FUNCTION_BLOCK xPPU_RFC
VAR_INPUT
	i_error: POINTER TO ErrorManager;
	i_process: POINTER TO ProcessManager;
	i_state: POINTER TO StateTracker;
END_VAR
VAR
	m_emptyParams: ParameterSet;
	m_subRes: EOperationResult;
	m_alarm_flags: ARRAY [1..10] OF BOOL := [FALSE, FALSE, FALSE, FALSE, FALSE, FALSE,FALSE, FALSE, FALSE, FALSE];
	m_delay200ms : TON;
	m_timer : TON;
	fb_RFC_WPAtStartFalling : F_TRIG;
	fb_RFC_WPAtEndFalling : F_TRIG;
	fb_RFC_WPAtEndReising : R_TRIG;
	m_timer_EndReset : TON; 

END_VAR

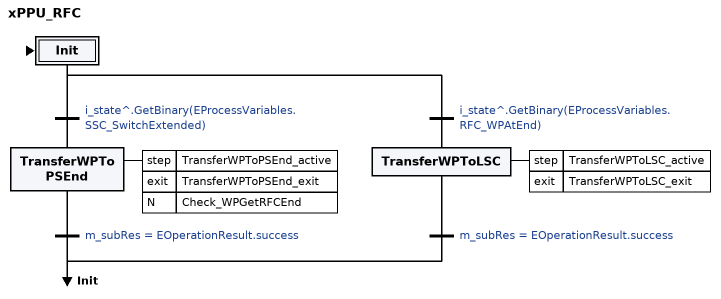
INITIAL_STEP Init:
END_STEP
TRANSITION FROM Init TO TransferWPToPSEnd
    := i_state^.GetBinary(EProcessVariables.SSC_SwitchExtended);
END_TRANSITION
STEP TransferWPToPSEnd:
    TransferWPToPSEnd_active(N);  // step action
    TransferWPToPSEnd_exit(P0);  // exit action
    Check_WPGetRFCEnd(N);
END_STEP
TRANSITION FROM TransferWPToPSEnd TO Init
    := m_subRes = EOperationResult.success;
END_TRANSITION
TRANSITION FROM Init TO TransferWPToLSC
    := i_state^.GetBinary(EProcessVariables.RFC_WPAtEnd);
END_TRANSITION
STEP TransferWPToLSC:
    TransferWPToLSC_active(N);  // step action
    TransferWPToLSC_exit(P0);  // exit action
END_STEP
TRANSITION FROM TransferWPToLSC TO Init
    := m_subRes = EOperationResult.success;
END_TRANSITION

ACTION Check_WPGetRFCEnd:
//new alarm
fb_RFC_WPAtStartFalling(CLK := i_state^.GetBinary(EProcessVariables.RFC_WPAtStart));
fb_RFC_WPAtEndFalling(CLK := i_state^.GetBinary(EProcessVariables.RFC_WPAtEnd));
fb_RFC_WPAtEndReising(CLK := i_state^.GetBinary(EProcessVariables.RFC_WPAtEnd));

// IF m_alarm_flags[1] = FALSE AND fb_RFC_WPAtStartFalling.Q 
//    AND NOT (i_state^.GetBinary(EProcessVariables.RFC_WPAtEnd))  
//    AND NOT fb_RFC_WPAtEndFalling.Q  
//    AND NOT fb_RFC_WPAtEndReising.Q   
// THEN
// 	i_error^.AddMessage(EAlarms.RFC_NotGetEnd, TRUE, ESeverity.error, 'WP in RFC can not get end from start');
//    	m_alarm_flags[1] := TRUE;
// 	m_timer (IN := m_alarm_flags[1], PT := T#1000MS);
// END_IF
// 
// IF m_timer.Q THEN
// 	fb_RFC_WPAtEndFalling(CLK := FALSE);
// 	fb_RFC_WPAtEndReising(CLK := FALSE);
// END_IF

IF fb_RFC_WPAtStartFalling.Q THEN
  m_timer_EndReset(IN := TRUE,PT := T#2S);
END_IF

IF i_state^.GetBinary(EProcessVariables.RFC_WPAtEnd) 
   OR fb_RFC_WPAtEndFalling.Q 
   OR fb_RFC_WPAtEndReising.Q 
THEN
  m_timer_EndReset(IN := FALSE);
END_IF

m_timer_EndReset();

IF (m_alarm_flags[1] = FALSE) 
   AND m_timer_EndReset.Q 
THEN
  i_error^.AddMessage(EAlarms.RFC_NotGetEnd, TRUE, ESeverity.error, 'WP in RFC can not get end from start');
  m_alarm_flags[1] := TRUE;
  m_timer_EndReset(IN := TRUE,PT := T#2S);
END_IF
END_ACTION

ACTION TransferWPToLSC_active:
m_subRes := i_process^.Execute(
	EBehaviorType.control_primitive,
	EPrimitives.RFC_TransferWorkpieceTo_LSC,
	m_emptyParams);
END_ACTION

ACTION TransferWPToLSC_exit:
i_state^.ShiftProduct(EProducts.RFC_product1, EProducts.LSC_product);

m_delay200ms(
  IN := TRUE,
  PT := T#200MS
);

IF m_delay200ms.Q THEN
  m_delay200ms(IN := FALSE);
i_state^.ShiftProduct(EProducts.RFC_product2, EProducts.LSC_product);
END_IF
END_ACTION

ACTION TransferWPToPSEnd_active:
m_subRes := i_process^.Execute(
	EBehaviorType.control_primitive,
	EPrimitives.RFC_TransferWorkpieceTo_PSEnd,
	m_emptyParams);
END_ACTION

ACTION TransferWPToPSEnd_exit:
m_alarm_flags[1] := FALSE; 
fb_RFC_WPAtEndFalling(CLK := FALSE);
fb_RFC_WPAtEndReising(CLK := FALSE);
END_ACTION

END_FUNCTION_BLOCK

(* stored: Version 1.1.0.1
   POU xPPU_RFC: Id {d90f6f73-9cc6-49aa-95fa-83b2098b3cd4}, SpecialFunc None
   Action Check_WPGetRFCEnd: Id {cce18ca6-d09f-4a59-a39d-e24a99227db3}
   Action TransferWPToLSC_active: Id {06822a62-8370-4767-a20c-06a31bc41e8d}
   Action TransferWPToLSC_exit: Id {47333ae5-1a92-4122-ac22-bb58dd1f2d05}
   Action TransferWPToPSEnd_active: Id {7486f9de-223c-4795-a1d2-77997eb33773}
   Action TransferWPToPSEnd_exit: Id {c0ddd4dc-ba68-4d56-8ade-908f3381b579} *)
